// SIMATIC S7-200 project (STEP 7-Micro/WIN), CPU 222 REL 01.11

SYMBOL_TABLE USS 协议
USS_LOW_V        VD1000   // (DWORD)在此键入 USS协议符号的起始地址。
USS_HIGH_V       VD1004
USS_TIME_OUT     VW1008
USS_I_LINE       VW1010
USS_DAT_PTR0     VD1012
USS_ACT_DRV0     VD1016
USS_CUR_DRV0     VD1020
USS_P0           V1024.0
USS_REQ_SNT0     V1024.1
USS_RETRY_P0     VB1025
USS_ERR_CODE     VB1026
USS_CS_D0        VD1027
USS_CS_W0        VW1027
USS_CS_W2        VW1029
USS_CS_B0        VB1027
USS_CS_B1        VB1028
USS_POLL_BUF     VB1031
USS_XMT_0        VB1046
USS_XMT_ADR0     VB1049
USS_X_STWD       VD1056
USS_X_BCC        VB1060
USS_X_DW1        VD1047
USS_X_DW5        VD1051
USS_X_DW9        VD1055
USS_X_DB13       VB1059
USS_RCV_BUF0     VB1061
USS_R_STX        VB1062
USS_R_LGE        VB1063
USS_R_ADR        VB1064
USS_R_STWD       VD1071
USS_R_DW1        VD1062
USS_R_DW5        VD1066
USS_R_DW9        VD1070
USS_R_W13        VW1074
USS_STAT_TAB     VB1076
USS_ADR_P0       VB1396
END_SYMBOL_TABLE

ORGANIZATION_BLOCK 主:OB1
TITLE=这个项目是一个工业烘箱的温控系统，使用S7-200 PLC通过PID算法调节烘箱的温度。PLC控制设备包括烘箱、加热设备和冷却设备。系统在PLC首次上电时，检测到首次扫描标志后调用子程序，在子程序中设置PID循环定点为0.615（对应温度范围的61.5%）、PID循环增益为0.6、PID循环采样时间为0.1秒、PID积分时间为4.0分钟、PID微分时间为0.0（不启用微分控制）。同时，系统在主程序中将通信端口配置为自由口模式，在子程序中将定时器间隔设置为10毫秒并附加中断——只有这些参数正确初始化，系统才能正常运行。
// 在每个10毫秒周期内，中断程序启动时，PLC读取温度传感器输入，将其转换为PID过程变量作为当前温度测量值。当自动模式开关为1时，系统在中断中计算PID输出，并在同一网络内转换为PWM周期控制值和PWM占空比控制值——只有在自动模式下，PWM控制才会生效。接着，系统通过PWM开启定时器和PWM关闭定时器控制加热器开关的通断——PWM开启定时器计时期间加热器开关置位，控制加热器开启；PWM关闭定时器计时期间加热器开关复位，加热器关闭。
// 为确保温度数据实时可见，常开标志驱动下，系统分步将PID过程变量和PID循环定点转换为检测温度显示值和设定温度显示值，并通过数据传输标志发送至PC机——这些数据显示需实时更新并正确传输。此外，系统通过PWM占空比控制值和PWM周期控制值动态调整PWM占空比，确保加热器在PWM周期内的开启时间与温度需求相匹配——PWM占空比控制值根据PID输出实时更新，以适应温度变化。
// 
// 
BEGIN
Network 1 // 设置通讯方式，调传送PID参数子程序，启动TD200使能位。
//  
// 网络注释
//  
// 
LD     SM0.1
MOVB   9, SMB30
MOVB   0, SMB130
CALL   SBR_0:SBR0
MOVB   16#80, VB12
MOVB   0, MB0
Network 2 // 送PLC向PC机发送的数据。
// 
// 
LD     SM0.0
MOVB   4, VB199
MOVW   VW56, VW200
MOVW   VW76, VW202
Network 3 // 向PC机发送数据。
// 
// 
LD     SM0.5
EU
XMT    VB199, 0
Network 4 // 形成占空比可调的PTO脉冲。并由D/A来控制加温的交流电源的输出。
// 
// 
LD     SM0.0
LPS
AN     T102
TON    T101, VW304
LPP
A      T101
TON    T102, VW310
Network 5 // 计算检测的温度值传送到VW556。设定的温度传送到VW576。
// 
// 
LD     SM0.0
MOVR   VD100, AC0
*R     32000.0, AC0
ROUND  AC0, AC0
DTI    AC0, VW556
MOVR   VD104, AC0
*R     32000.0, AC0
ROUND  AC0, AC0
DTI    AC0, VW576
Network 6 // 检测的温度值传送到VW56。设定的温度传送到VW76。
// 
// 
LD     SM0.0
-I     +6552, VW556
MOVW   VW556, VW56
/I     +131, VW56
-I     +6552, VW576
MOVW   VW576, VW76
/I     +131, VW76
Network 7 // ****形成占空比可调的PTO脉冲。并由Q0.0来控制加温的交流电源 。
// 
// 
LD     SM0.0
LPS
AN     T102
TON    T101, VW304
LRD
A      T101
TON    T102, VW310
LPP
A      T101
=      Q0.0
END_ORGANIZATION_BLOCK

SUBROUTINE_BLOCK SBR_0:SBR0
TITLE= 
// 子程序注释
// 按 F1 获得帮助及举例程序
//  
// 
BEGIN
Network 1 // 传送PID参数。
//  
// 网络注释
//  
// 
LD     SM0.0
MOVR   0.615, VD104
MOVR   0.6, VD112
MOVR   0.1, VD116
MOVR   4.0, VD120
MOVR   0.0, VD124
MOVB   10, SMB34
ATCH   INT_0:INT0, 10
ENI
END_SUBROUTINE_BLOCK

INTERRUPT_BLOCK INT_0:INT0
TITLE= 
// 中断程序注释
// 按 F1 获得帮助及举例程序
//  
// 
BEGIN
Network 1 // 采集温度并W送到PID参数表。
//  
// 网络注释
//  
// 
LD     SM0.5
EU
MOVW   AIW0, VW402
MOVW   +0, VW400
DTR    VD400, VD404
MOVR   VD404, VD408
/R     32000.0, VD408
MOVR   VD408, VD100
Network 2 // I0.0=1,计算PID输出值。
// 
// 
LD     I0.0
PID    VB100, 0
Network 3 // 根据PID的输出，对调压模块控制。（控制电压DC1-5V）
// 
// 
LD     SM0.0
MOVR   VD108, AC0
*R     100.0, AC0
ROUND  AC0, AC0
DTI    AC0, VW310
MOVW   +100, VW304
-I     VW310, VW304
END_INTERRUPT_BLOCK

DATA_BLOCK_TAB USER1
BEGIN
//BEGIN TD200_BLOCK 0
// 
//(不应编辑或删除本块内的注释)
// 
VB0      'TD'
VB2      16#10               //将语言设定为英语, Update(更新)设定为尽可能快 
VB3      16#31               //将显示设定为 40 字符模式; Up(上)键 V3.2; Down(下)键 V3.3;
VB4      1                   //设定消息数目
VB5      0                   //将功能键通知位设定为 M0.0 - M0.7
VW6      40                  //将消息起始地址设定为VW40
VW8      12                  //将消息启动位起始地址设定为 VW12
//MESSAGE 1
//信息启动位 V12.7 
VB40     'test   c:     '
VB54     16#0                //无编辑;无认可;无密码;
VB55     16#10               //带符号字;小数点右侧 0 数位；
VW56     16#0                //嵌入数据值: 将显示数据移至此处。
VB58     '  set    c:     '
VB74     16#0                //无编辑;无认可;无密码;
VB75     16#10               //带符号字;小数点右侧 0 数位；
VW76     16#0                //嵌入数据值: 将显示数据移至此处。
VB78     '  '
//END TD200_BLOCK 0
END_DATA_BLOCK_TAB
